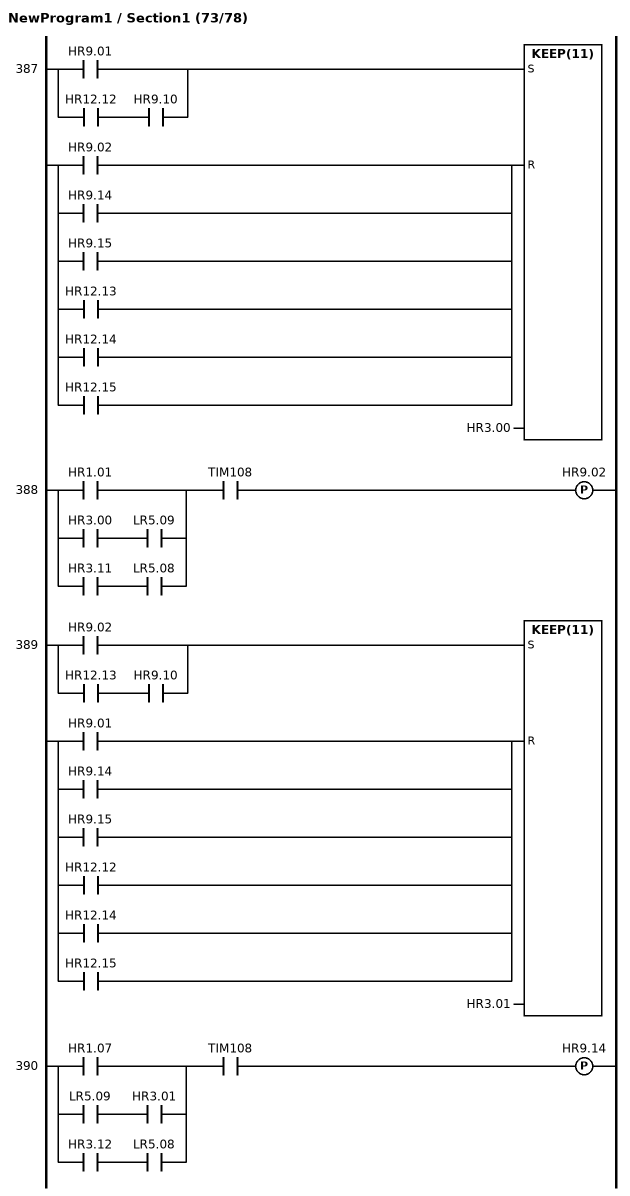
; [picture p72: NewProgram1 / Section1, rungs 387-390]
; rung 387
LD HR9.01
LD HR12.12
AND HR9.10
ORLD
LD HR9.02
OR HR9.14
OR HR9.15
OR HR12.13
OR HR12.14
OR HR12.15
KEEP(11) HR3.00
; rung 388
LD HR1.01
LD HR3.00
AND LR5.09
ORLD
LD HR3.11
AND LR5.08
ORLD
AND TIM108
DIFU(13) HR9.02
; rung 389
LD HR9.02
LD HR12.13
AND HR9.10
ORLD
LD HR9.01
OR HR9.14
OR HR9.15
OR HR12.12
OR HR12.14
OR HR12.15
KEEP(11) HR3.01
; rung 390
LD HR1.07
LD LR5.09
AND HR3.01
ORLD
LD HR3.12
AND LR5.08
ORLD
AND TIM108
DIFU(13) HR9.14

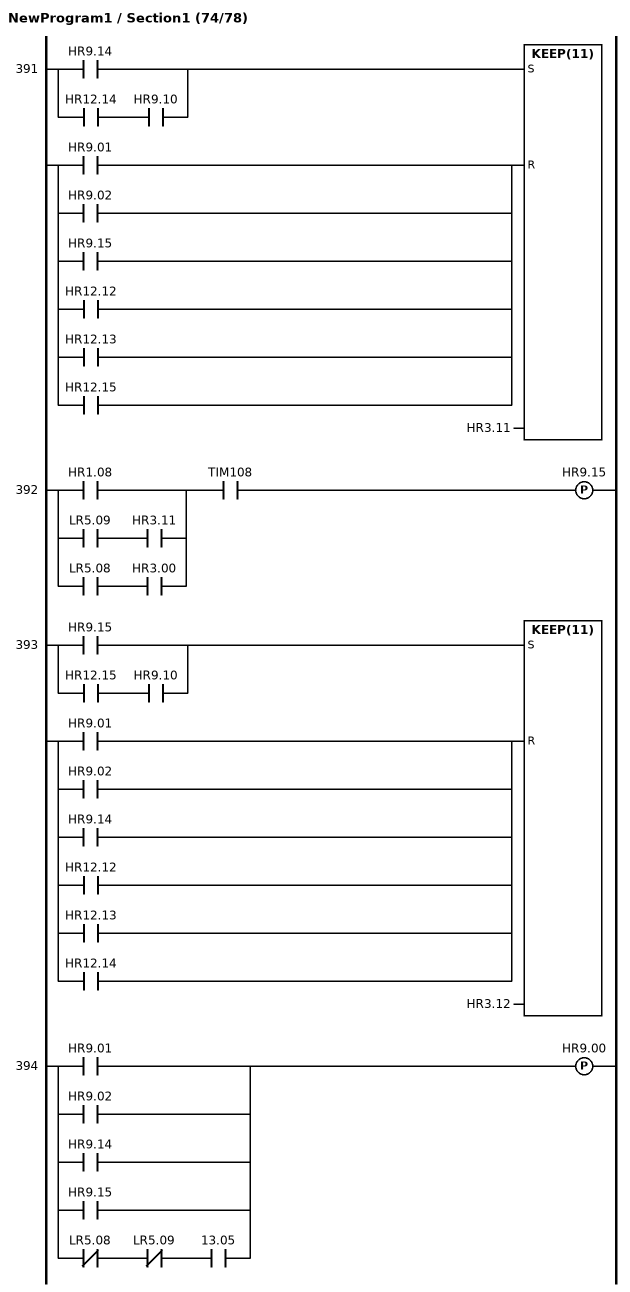
; rung 391
LD HR9.14
LD HR12.14
AND HR9.10
ORLD
LD HR9.01
OR HR9.02
OR HR9.15
OR HR12.12
OR HR12.13
OR HR12.15
KEEP(11) HR3.11
; rung 392
LD HR1.08
LD LR5.09
AND HR3.11
ORLD
LD LR5.08
AND HR3.00
ORLD
AND TIM108
DIFU(13) HR9.15
; rung 393
LD HR9.15
LD HR12.15
AND HR9.10
ORLD
LD HR9.01
OR HR9.02
OR HR9.14
OR HR12.12
OR HR12.13
OR HR12.14
KEEP(11) HR3.12
; rung 394
LD HR9.01
OR HR9.02
OR HR9.14
OR HR9.15
LDNOT LR5.08
ANDNOT LR5.09
AND 13.05
ORLD
DIFU(13) HR9.00

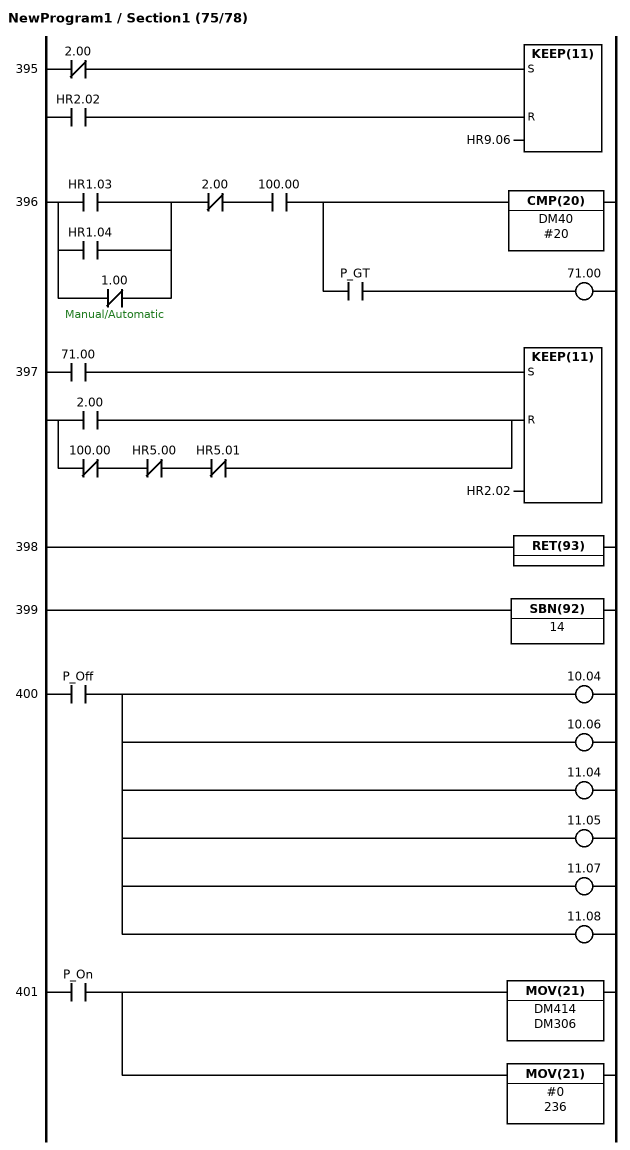
; rung 395
LDNOT 2.00
LD HR2.02
KEEP(11) HR9.06
; rung 396
LD HR1.03
OR HR1.04
ORNOT 1.00  ; Manual/Automatic
ANDNOT 2.00
AND 100.00
CMP(20) DM40 #20
AND P_GT
OUT 71.00
; rung 397
LD 71.00
LD 2.00
LDNOT 100.00
ANDNOT HR5.00
ANDNOT HR5.01
ORLD
KEEP(11) HR2.02
; rung 398
RET(93)
; rung 399
SBN(92) 14
; rung 400
LD P_Off
OUT 10.04
OUT 10.06
OUT 11.04
OUT 11.05
OUT 11.07
OUT 11.08
; rung 401
LD P_On
MOV(21) DM414 DM306
MOV(21) #0 236

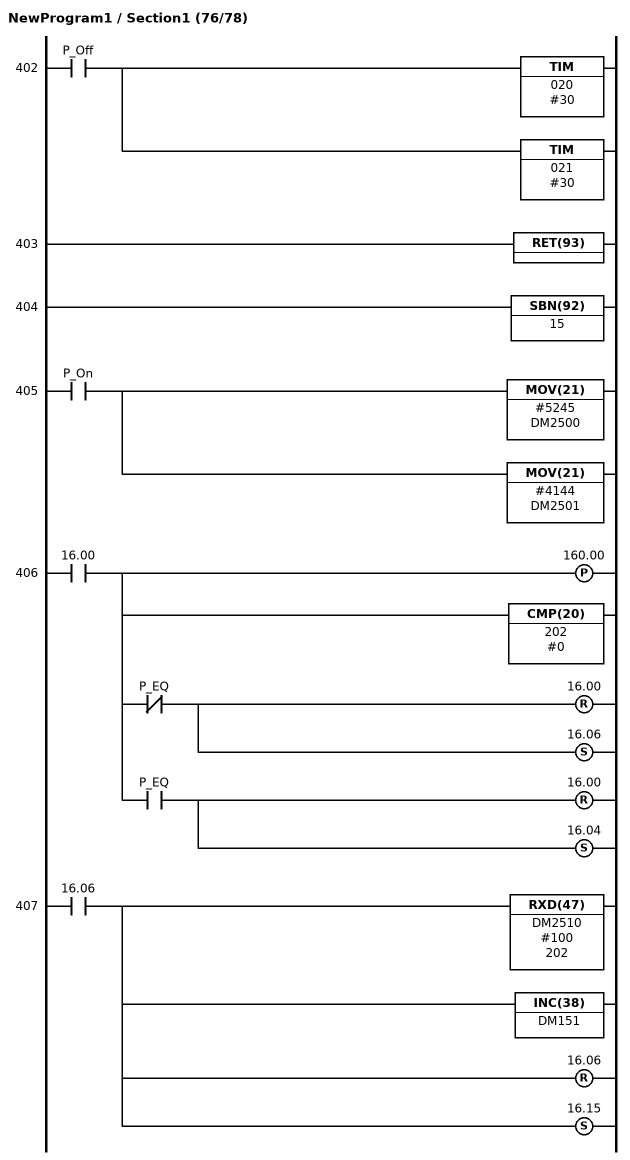
; rung 402
LD P_Off
TIM 020 #30
TIM 021 #30
; rung 403
RET(93)
; rung 404
SBN(92) 15
; rung 405
LD P_On
MOV(21) #5245 DM2500
MOV(21) #4144 DM2501
; rung 406
LD 16.00
OUT TR0
DIFU(13) 160.00
CMP(20) 202 #0
ANDNOT P_EQ
RSET 16.00
SET 16.06
LD TR0
AND P_EQ
RSET 16.00
SET 16.04
; rung 407
LD 16.06
RXD(47) DM2510 #100 202
INC(38) DM151
RSET 16.06
SET 16.15

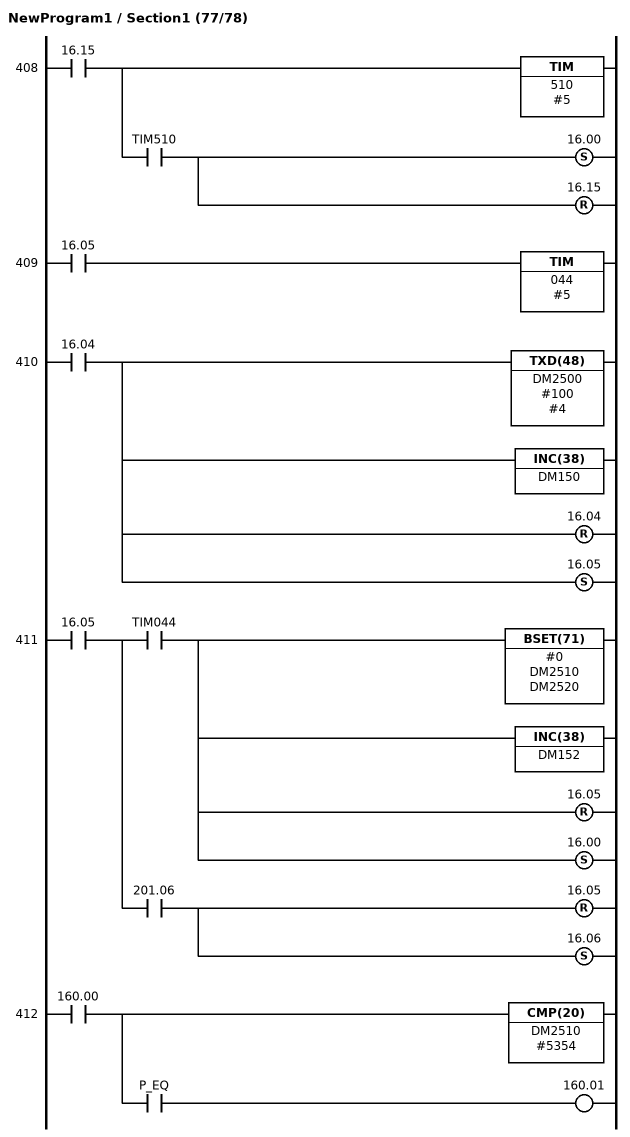
; rung 408
LD 16.15
TIM 510 #5
AND TIM510
SET 16.00
RSET 16.15
; rung 409
LD 16.05
TIM 044 #5
; rung 410
LD 16.04
TXD(48) DM2500 #100 #4
INC(38) DM150
RSET 16.04
SET 16.05
; rung 411
LD 16.05
OUT TR0
AND TIM044
BSET(71) #0 DM2510 DM2520
INC(38) DM152
RSET 16.05
SET 16.00
LD TR0
AND 201.06
RSET 16.05
SET 16.06
; rung 412
LD 160.00
CMP(20) DM2510 #5354
AND P_EQ
OUT 160.01

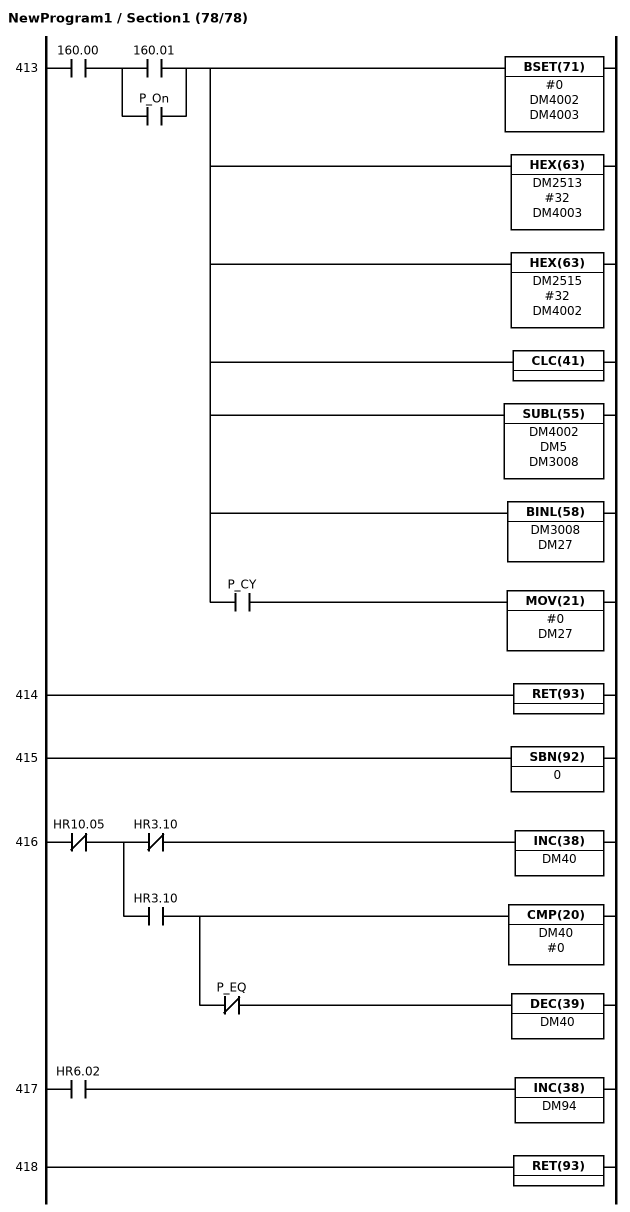
; rung 413
LD 160.00
LD 160.01
OR P_On
ANDLD
BSET(71) #0 DM4002 DM4003
HEX(63) DM2513 #32 DM4003
HEX(63) DM2515 #32 DM4002
CLC(41)
SUBL(55) DM4002 DM5 DM3008
BINL(58) DM3008 DM27
AND P_CY
MOV(21) #0 DM27
; rung 414
RET(93)
; rung 415
SBN(92) 0
; rung 416
LDNOT HR10.05
OUT TR0
ANDNOT HR3.10
INC(38) DM40
LD TR0
AND HR3.10
CMP(20) DM40 #0
ANDNOT P_EQ
DEC(39) DM40
; rung 417
LD HR6.02
INC(38) DM94
; rung 418
RET(93)
; rung 419
END(01)